Universal Robots PolyScope program: a_to_d.urp

Program a_to_d (installation=string_planes directory=/programs/string_crossings createdIn=5.17.3 lastSavedIn=5.17.3 robotSerialNumber=20245501435)
Calibrated DH parameters: a=[0.000154, -0.137004, -0.385524, -0.00002, 0.000092, 0]; d=[0.162441, 211.794786, -230.585024, 18.923638, 0.099786, 0.09951]; alpha=[1.569493, -0.001902, 0.003874, 1.570111, -1.570167, 0]; deltaTheta=[0, -1.242934, 1.056292, 0.186646, 0.000002, 0.000001]
InitVariablesNode
Robot Program (runOnlyOnce=true)
  bow_section := -1
  If bow_section≟-1
    MoveJ speed 60 deg/s, acceleration 80 deg/s^2 (useActiveTCP=true) feature=Base
      Waypoint Waypoint_7 (Relative): relativeFromPosition TCP in base x=277.235 y=734.032 z=156.893 mm, rx=1.7389 ry=2.3104 rz=-1.1077 rad; joints [-126.647, -28.124, 54.729, -74.617, -91.964, -141.812] deg; TCP offset x=28.21 y=-96.107 z=-99.69 mm, rx=0 ry=0 rz=0 rad; TCP in base x=316.092 y=723.606 z=117.8 mm, rx=-1.5349 ry=-2.2386 rz=1.1274 rad; joints [-128.46, -21.869, 50.821, -72.931, -81.953, -152.855] deg
  ElseIf bow_section≟0
    MoveJ speed 60 deg/s, acceleration 80 deg/s^2 (useActiveTCP=true) feature=Base
      Waypoint Waypoint_1 (Relative): relativeFromPosition TCP in base x=327.074 y=542.849 z=231.417 mm, rx=1.6821 ry=2.3247 rz=-1.1115 rad; joints [-139.55, -50.207, 85.865, -84.66, -102.289, -153.001] deg; TCP in base x=329.632 y=457.693 z=123.027 mm, rx=-1.5368 ry=-2.1747 rz=1.1049 rad; joints [-145.135, -44.399, 100.427, -98.676, -90.572, -164.15] deg
  Else 
    MoveJ speed 60 deg/s, acceleration 80 deg/s^2 (useActiveTCP=true) feature=Base
      Waypoint Waypoint_2 (Relative): relativeFromPosition TCP in base x=374.965 y=359.133 z=303.036 mm, rx=1.6274 ry=2.3373 rz=-1.1146 rad; joints [-156.116, -66.368, 101.551, -88.734, -114.43, -168.118] deg; TCP in base x=340.8 y=238.63 z=127.345 mm, rx=-1.5375 ry=-2.1223 rz=1.0863 rad; joints [-167.853, -53.47, 123.568, -113.68, -104.544, -179.466] deg
